FUNCTION_BLOCK SystemBundle
VAR_INPUT
END_VAR
VAR_OUTPUT
END_VAR
VAR
	_timeProvider		: TimeProvider;
END_VAR

METHOD Call : BOOL
VAR_INPUT
END_VAR

_timeProvider();
END_METHOD


METHOD GetTaskHeartbeat : BOOL
VAR_INPUT
END_VAR

GetTaskHeartbeat := TaskHeartbeat(update := FALSE);
END_METHOD

PROPERTY TimeProvider : REFERENCE TO TimeProvider
GET

TimeProvider REF= _timeProvider;
END_GET
END_PROPERTY

END_FUNCTION_BLOCK

(* stored: Version 1.1.0.1, ProductVersion 3.1.4024.12
   POU SystemBundle: Id {cfe906a7-cb4d-49b4-a6a1-3e9b01fb4a45}, SpecialFunc None
   Method Call: Id {a86f7c66-f1a5-4ec2-a690-f1af2a631b65}
   Method GetTaskHeartbeat: Id {919fd3d0-2e58-4a8a-97d4-6abedb9132b7}
   Property TimeProvider: Id {4ff49010-98e8-4db2-a0eb-45c0a43fd21f}
   Get Get: Id {4df5db3e-22e7-4af9-a3e4-1d803909c512} *)
